REGION Network 12
   // 读重量
   RUNG wire#powerrail
      #Modbus_Master.Modbus_Master(REQ := wire#w1, MB_ADDR := 3, MODE :=, DATA_ADDR := 40104, DATA_LEN := 2, DATA_PTR := #ST6, DONE =>, BUSY =>, ERROR =>, STATUS =>)
      Move(in := #ST6[0], out1 => #B管道内径AT[1])
      Move(in := #ST6[1], out1 => #B管道内径AT[0])
   END_RUNG
   RUNG wire#powerrail
      { S7_Templates := "SrcType := Int" } EQ_Contact(in1 := #CTU.CV, in2 := 8)
      P_Trig( #TP[8] )
   END_RUNG wire#w1
   // the same network as SCL:
   #_w1 := #CTU.CV = 8;
   #_w2 := #_w1 AND NOT #TP[8];   // rising edge
   #TP[8] := #_w1;
   #Modbus_Master(REQ := #_w2, MB_ADDR := 3, DATA_ADDR := 40104, DATA_LEN := 2, DATA_PTR := #ST6, ENO => #_w3);   // Modbus_Master
   IF #_w3 THEN
       #B管道内径AT[1] := #ST6[0];
       #B管道内径AT[0] := #ST6[1];
   END_IF;
END_REGION
END_FUNCTION_BLOCK

FUNCTION_BLOCK "通信心跳"   // FB46, LAD
{ S7_Optimized_Access := 'TRUE' }
VERSION : 0.1
// stored: AutoNumber true, IsIECCheckEnabled false, IsRetainMemResEnabled false, MemoryReserve 100, SetENOAutomatically false, UDAEnableTagReadback false
   VAR_OUTPUT
      通信失联 : Bool;
   END_VAR
   VAR_IN_OUT
      real_SC输出值 : Real;
      real_FK反馈值 : Real;
      超时时间 : Time := T#30S;
      i : Int;
   END_VAR
   VAR
      t1 : TON_TIME;
      t2 { S7_SetPoint := 'True'} : TON_TIME;
      RT1 : R_TRIG;
      间隔时间 : Time := T#5S;
      SC输出值 : Int;
      FK反馈值 : Int;
   END_VAR
   VAR_TEMP
      TM_FZ : Int;
   END_VAR
BEGIN

REGION Network 2 (SCL)
   // 间隔时间，通针开关
   #TM_FZ:=#FK反馈值;

   #SC输出值 := REAL_TO_INT(#real_SC输出值);
   #FK反馈值 := REAL_TO_INT(#real_FK反馈值);

   #t1(IN := (#TM_FZ <> #SC输出值) ,
       PT := #超时时间,
       Q=>#通信失联);


   (* IF #t1.Q THEN
       (* #TM_FZ := 1; *)
       #SC输出值 := #SC输出值 - 1;
   END_IF; *)

   IF #TM_FZ =#SC输出值 THEN

       IF #SC输出值 MOD 2 =0 THEN

           #SC输出值 := #SC输出值 + 1;
       ELSE

           #SC输出值 := #SC输出值 - 1;
       END_IF;

   END_IF;
END_REGION
END_FUNCTION_BLOCK

FUNCTION_BLOCK "52普通脉冲"   // FB23, SCL
{ S7_Optimized_Access := 'TRUE' }
VERSION : 0.1
// stored: AutoNumber true, IsIECCheckEnabled false, IsRetainMemResEnabled false, MemoryReserve 100, SetENOAutomatically false, UDAEnableTagReadback false
   VAR_INPUT
      模式设定 : Real;
      QD : Bool;
      On_Time : Real;
      Stop_Time : Real;
      Num : Int;
   END_VAR
   VAR_OUTPUT
      Output_1 : Bool;
      Output_2 : Bool;
      Output_3 : Bool;
      Output_4 : Bool;
      Output_5 : Bool;
      Output_6 : Bool;
      Output_7 : Bool;
      Output_8 : Bool;
      Num_now : Int;
   END_VAR
   VAR
      Stoptime : Time;
      WorkTime : Time;
      TON_ON : Array[1..10] of TON_TIME;
      TON_OFF : Array[1..10] of TON_TIME;
   END_VAR
BEGIN

   IF #模式设定 = 1.0  OR #模式设定 = 2.0  THEN
       #Stoptime := DINT_TO_TIME(REAL_TO_DINT(#Stop_Time * 1000.0));
       //#WorkTime := DINT_TO_TIME(REAL_TO_DINT(#On_Time * 1000));
        #WorkTime := REAL_TO_DINT(#On_Time);

       IF NOT #QD THEN
           #Num_now := 0;
       ELSE

           IF #Num <= 8 THEN
               #Num_now := #Num;
           ELSE
               #Num_now := 8;
           END_IF;

       END_IF;



       CASE #Num_now OF
           1:
               #TON_ON[1](IN := #QD AND NOT #TON_OFF[1].Q,
                          PT := #WorkTime);
               #TON_OFF[1](IN := #QD AND #TON_ON[1].Q,
                           PT := #Stoptime);


               #Output_1 := #QD AND NOT #TON_ON[1].Q;


           2:  // Statement section case 1
               #TON_ON[1](IN := #QD AND NOT #TON_OFF[2].Q,
                          PT := #WorkTime);
               #TON_OFF[1](IN := #QD AND #TON_ON[1].Q,
                           PT := #Stoptime);
               #TON_ON[2](IN := #QD AND #TON_ON[1].Q AND #TON_OFF[1].Q,
                          PT := #WorkTime);
               #TON_OFF[2](IN := #QD AND #TON_ON[1].Q AND #TON_OFF[1].Q AND #TON_ON[2].Q,
                           PT := #Stoptime);

               #Output_1 := #QD AND NOT #TON_ON[1].Q;
               #Output_2 := #QD AND #TON_ON[1].Q AND #TON_OFF[1].Q AND NOT #TON_ON[2].Q;

           3:  // Statement section case 2 to 4
               #TON_ON[1](IN := #QD AND NOT #TON_OFF[3].Q,
                          PT := #WorkTime);
               #TON_OFF[1](IN := #QD AND #TON_ON[1].Q,
                           PT := #Stoptime);
               #TON_ON[2](IN := #QD AND #TON_ON[1].Q AND #TON_OFF[1].Q,
                          PT := #WorkTime);
               #TON_OFF[2](IN := #QD AND #TON_ON[1].Q AND #TON_OFF[1].Q AND #TON_ON[2].Q,
                           PT := #Stoptime);
               #TON_ON[3](IN := #QD AND #TON_ON[1].Q AND #TON_OFF[1].Q AND #TON_ON[2].Q AND #TON_OFF[2].Q,
                          PT := #WorkTime);
               #TON_OFF[3](IN := #QD AND #TON_ON[1].Q AND #TON_OFF[1].Q AND #TON_ON[2].Q AND #TON_OFF[2].Q AND #TON_ON[3].Q,
                           PT := #Stoptime);
               #Output_1 := #QD AND NOT #TON_ON[1].Q;
               #Output_2 := #QD AND #TON_ON[1].Q AND #TON_OFF[1].Q AND NOT #TON_ON[2].Q;
               #Output_3 := #QD AND #TON_ON[1].Q AND #TON_OFF[1].Q AND #TON_ON[2].Q AND #TON_OFF[2].Q AND NOT #TON_ON[3].Q;
           4:  // Statement section case 2 to 4
               #TON_ON[1](IN := #QD AND NOT #TON_OFF[4].Q,
                          PT := #WorkTime);
               #TON_OFF[1](IN := #QD AND #TON_ON[1].Q,
                           PT := #Stoptime);
               #TON_ON[2](IN := #QD AND #TON_ON[1].Q AND #TON_OFF[1].Q,
                          PT := #WorkTime);
               #TON_OFF[2](IN := #QD AND #TON_ON[1].Q AND #TON_OFF[1].Q AND #TON_ON[2].Q,
                           PT := #Stoptime);
               #TON_ON[3](IN := #QD AND #TON_ON[1].Q AND #TON_OFF[1].Q AND #TON_ON[2].Q AND #TON_OFF[2].Q,
                          PT := #WorkTime);
               #TON_OFF[3](IN := #QD AND #TON_ON[1].Q AND #TON_OFF[1].Q AND #TON_ON[2].Q AND #TON_OFF[2].Q AND #TON_ON[3].Q,
                           PT := #Stoptime);

               #TON_ON[4](IN := #QD AND #TON_ON[1].Q AND #TON_OFF[1].Q AND #TON_ON[2].Q AND #TON_OFF[2].Q AND #TON_ON[3].Q AND #TON_OFF[3].Q,
                          PT := #WorkTime);
               #TON_OFF[4](IN := #QD AND #TON_ON[1].Q AND #TON_OFF[1].Q AND #TON_ON[2].Q AND #TON_OFF[2].Q AND #TON_ON[3].Q AND #TON_OFF[3].Q AND #TON_ON[4].Q,
                           PT := #Stoptime);


               #Output_1 := #QD AND NOT #TON_ON[1].Q;
               #Output_2 := #QD AND #TON_ON[1].Q AND #TON_OFF[1].Q AND NOT #TON_ON[2].Q;
               #Output_3 := #QD AND #TON_ON[1].Q AND #TON_OFF[1].Q AND #TON_ON[2].Q AND #TON_OFF[2].Q AND NOT #TON_ON[3].Q;
               #Output_4 := #QD AND #TON_ON[1].Q AND #TON_OFF[1].Q AND #TON_ON[2].Q AND #TON_OFF[2].Q AND #TON_ON[3].Q AND #TON_OFF[3].Q AND NOT #TON_ON[4].Q;

           5:  // Statement section case 2 to 4
               #TON_ON[1](IN := #QD AND NOT #TON_OFF[5].Q,
                          PT := #WorkTime);
               #TON_OFF[1](IN := #QD AND #TON_ON[1].Q,
                           PT := #Stoptime);
               #TON_ON[2](IN := #QD AND #TON_ON[1].Q AND #TON_OFF[1].Q,
                          PT := #WorkTime);
               #TON_OFF[2](IN := #QD AND #TON_ON[1].Q AND #TON_OFF[1].Q AND #TON_ON[2].Q,
                           PT := #Stoptime);
               #TON_ON[3](IN := #QD AND #TON_ON[1].Q AND #TON_OFF[1].Q AND #TON_ON[2].Q AND #TON_OFF[2].Q,
                          PT := #WorkTime);
               #TON_OFF[3](IN := #QD AND #TON_ON[1].Q AND #TON_OFF[1].Q AND #TON_ON[2].Q AND #TON_OFF[2].Q AND #TON_ON[3].Q,
                           PT := #Stoptime);

               #TON_ON[4](IN := #QD AND #TON_ON[1].Q AND #TON_OFF[1].Q AND #TON_ON[2].Q AND #TON_OFF[2].Q AND #TON_ON[3].Q AND #TON_OFF[3].Q,
                          PT := #WorkTime);
               #TON_OFF[4](IN := #QD AND #TON_ON[1].Q AND #TON_OFF[1].Q AND #TON_ON[2].Q AND #TON_OFF[2].Q AND #TON_ON[3].Q AND #TON_OFF[3].Q AND #TON_ON[4].Q,
                           PT := #Stoptime);

               #TON_ON[5](IN := #QD AND #TON_ON[1].Q AND #TON_OFF[1].Q AND #TON_ON[2].Q AND #TON_OFF[2].Q AND #TON_ON[3].Q AND #TON_OFF[3].Q AND #TON_ON[4].Q AND #TON_OFF[4].Q,
                          PT := #WorkTime);
               #TON_OFF[5](IN := #QD AND #TON_ON[1].Q AND #TON_OFF[1].Q AND #TON_ON[2].Q AND #TON_OFF[2].Q AND #TON_ON[3].Q AND #TON_OFF[3].Q AND #TON_ON[4].Q AND #TON_OFF[4].Q AND #TON_ON[5].Q,
                           PT := #Stoptime);


               #Output_1 := #QD AND NOT #TON_ON[1].Q;
               #Output_2 := #QD AND #TON_ON[1].Q AND #TON_OFF[1].Q AND NOT #TON_ON[2].Q;
               #Output_3 := #QD AND #TON_ON[1].Q AND #TON_OFF[1].Q AND #TON_ON[2].Q AND #TON_OFF[2].Q AND NOT #TON_ON[3].Q;
               #Output_4 := #QD AND #TON_ON[1].Q AND #TON_OFF[1].Q AND #TON_ON[2].Q AND #TON_OFF[2].Q AND #TON_ON[3].Q AND #TON_OFF[3].Q AND NOT #TON_ON[4].Q;
               #Output_5 := #QD AND #TON_ON[1].Q AND #TON_OFF[1].Q AND #TON_ON[2].Q AND #TON_OFF[2].Q AND #TON_ON[3].Q AND #TON_OFF[3].Q AND #TON_ON[4].Q AND #TON_OFF[4].Q AND NOT #TON_ON[5].Q;

           6:  // Statement section case 2 to 4
               #TON_ON[1](IN := #QD AND NOT #TON_OFF[6].Q,
                          PT := #WorkTime);
               #TON_OFF[1](IN := #QD AND #TON_ON[1].Q,
                           PT := #Stoptime);
               #TON_ON[2](IN := #QD AND #TON_ON[1].Q AND #TON_OFF[1].Q,
                          PT := #WorkTime);
               #TON_OFF[2](IN := #QD AND #TON_ON[1].Q AND #TON_OFF[1].Q AND #TON_ON[2].Q,
                           PT := #Stoptime);
               #TON_ON[3](IN := #QD AND #TON_ON[1].Q AND #TON_OFF[1].Q AND #TON_ON[2].Q AND #TON_OFF[2].Q,
                          PT := #WorkTime);
               #TON_OFF[3](IN := #QD AND #TON_ON[1].Q AND #TON_OFF[1].Q AND #TON_ON[2].Q AND #TON_OFF[2].Q AND #TON_ON[3].Q,
                           PT := #Stoptime);

               #TON_ON[4](IN := #QD AND #TON_ON[1].Q AND #TON_OFF[1].Q AND #TON_ON[2].Q AND #TON_OFF[2].Q AND #TON_ON[3].Q AND #TON_OFF[3].Q,
                          PT := #WorkTime);
               #TON_OFF[4](IN := #QD AND #TON_ON[1].Q AND #TON_OFF[1].Q AND #TON_ON[2].Q AND #TON_OFF[2].Q AND #TON_ON[3].Q AND #TON_OFF[3].Q AND #TON_ON[4].Q,
                           PT := #Stoptime);

               #TON_ON[5](IN := #QD AND #TON_ON[1].Q AND #TON_OFF[1].Q AND #TON_ON[2].Q AND #TON_OFF[2].Q AND #TON_ON[3].Q AND #TON_OFF[3].Q AND #TON_ON[4].Q AND #TON_OFF[4].Q,
                          PT := #WorkTime);
               #TON_OFF[5](IN := #QD AND #TON_ON[1].Q AND #TON_OFF[1].Q AND #TON_ON[2].Q AND #TON_OFF[2].Q AND #TON_ON[3].Q AND #TON_OFF[3].Q AND #TON_ON[4].Q AND #TON_OFF[4].Q AND #TON_ON[5].Q,
                           PT := #Stoptime);

               #TON_ON[6](IN := #QD AND #TON_ON[1].Q AND #TON_OFF[1].Q AND #TON_ON[2].Q AND #TON_OFF[2].Q AND #TON_ON[3].Q AND #TON_OFF[3].Q AND #TON_ON[4].Q AND #TON_OFF[4].Q AND #TON_ON[5].Q AND #TON_OFF[5].Q,
                          PT := #WorkTime);
               #TON_OFF[6](IN := #QD AND #TON_ON[1].Q AND #TON_OFF[1].Q AND #TON_ON[2].Q AND #TON_OFF[2].Q AND #TON_ON[3].Q AND #TON_OFF[3].Q AND #TON_ON[4].Q AND #TON_OFF[4].Q AND #TON_ON[5].Q AND #TON_OFF[5].Q AND #TON_ON[6].Q,
                           PT := #Stoptime);


               #Output_1 := #QD AND NOT #TON_ON[1].Q;
               #Output_2 := #QD AND #TON_ON[1].Q AND #TON_OFF[1].Q AND NOT #TON_ON[2].Q;
               #Output_3 := #QD AND #TON_ON[1].Q AND #TON_OFF[1].Q AND #TON_ON[2].Q AND #TON_OFF[2].Q AND NOT #TON_ON[3].Q;
               #Output_4 := #QD AND #TON_ON[1].Q AND #TON_OFF[1].Q AND #TON_ON[2].Q AND #TON_OFF[2].Q AND #TON_ON[3].Q AND #TON_OFF[3].Q AND NOT #TON_ON[4].Q;
               #Output_5 := #QD AND #TON_ON[1].Q AND #TON_OFF[1].Q AND #TON_ON[2].Q AND #TON_OFF[2].Q AND #TON_ON[3].Q AND #TON_OFF[3].Q AND #TON_ON[4].Q AND #TON_OFF[4].Q AND NOT #TON_ON[5].Q;
               #Output_6 := #QD AND #TON_ON[1].Q AND #TON_OFF[1].Q AND #TON_ON[2].Q AND #TON_OFF[2].Q AND #TON_ON[3].Q AND #TON_OFF[3].Q AND #TON_ON[4].Q AND #TON_OFF[4].Q AND #TON_ON[5].Q AND #TON_OFF[5].Q AND NOT #TON_ON[6].Q;

           7:  // Statement section case 2 to 4
               #TON_ON[1](IN := #QD AND NOT #TON_OFF[7].Q,
                          PT := #WorkTime);
               #TON_OFF[1](IN := #QD AND #TON_ON[1].Q,
                           PT := #Stoptime);
               #TON_ON[2](IN := #QD AND #TON_ON[1].Q AND #TON_OFF[1].Q,
                          PT := #WorkTime);
               #TON_OFF[2](IN := #QD AND #TON_ON[1].Q AND #TON_OFF[1].Q AND #TON_ON[2].Q,
                           PT := #Stoptime);
               #TON_ON[3](IN := #QD AND #TON_ON[1].Q AND #TON_OFF[1].Q AND #TON_ON[2].Q AND #TON_OFF[2].Q,
                          PT := #WorkTime);
               #TON_OFF[3](IN := #QD AND #TON_ON[1].Q AND #TON_OFF[1].Q AND #TON_ON[2].Q AND #TON_OFF[2].Q AND #TON_ON[3].Q,
                           PT := #Stoptime);

               #TON_ON[4](IN := #QD AND #TON_ON[1].Q AND #TON_OFF[1].Q AND #TON_ON[2].Q AND #TON_OFF[2].Q AND #TON_ON[3].Q AND #TON_OFF[3].Q,
                          PT := #WorkTime);
               #TON_OFF[4](IN := #QD AND #TON_ON[1].Q AND #TON_OFF[1].Q AND #TON_ON[2].Q AND #TON_OFF[2].Q AND #TON_ON[3].Q AND #TON_OFF[3].Q AND #TON_ON[4].Q,
                           PT := #Stoptime);

               #TON_ON[5](IN := #QD AND #TON_ON[1].Q AND #TON_OFF[1].Q AND #TON_ON[2].Q AND #TON_OFF[2].Q AND #TON_ON[3].Q AND #TON_OFF[3].Q AND #TON_ON[4].Q AND #TON_OFF[4].Q,
                          PT := #WorkTime);
               #TON_OFF[5](IN := #QD AND #TON_ON[1].Q AND #TON_OFF[1].Q AND #TON_ON[2].Q AND #TON_OFF[2].Q AND #TON_ON[3].Q AND #TON_OFF[3].Q AND #TON_ON[4].Q AND #TON_OFF[4].Q AND #TON_ON[5].Q,
                           PT := #Stoptime);

               #TON_ON[6](IN := #QD AND #TON_ON[1].Q AND #TON_OFF[1].Q AND #TON_ON[2].Q AND #TON_OFF[2].Q AND #TON_ON[3].Q AND #TON_OFF[3].Q AND #TON_ON[4].Q AND #TON_OFF[4].Q AND #TON_ON[5].Q AND #TON_OFF[5].Q,
                          PT := #WorkTime);
               #TON_OFF[6](IN := #QD AND #TON_ON[1].Q AND #TON_OFF[1].Q AND #TON_ON[2].Q AND #TON_OFF[2].Q AND #TON_ON[3].Q AND #TON_OFF[3].Q AND #TON_ON[4].Q AND #TON_OFF[4].Q AND #TON_ON[5].Q AND #TON_OFF[5].Q AND #TON_ON[6].Q,
                           PT := #Stoptime);

               #TON_ON[7](IN := #QD AND #TON_ON[1].Q AND #TON_OFF[1].Q AND #TON_ON[2].Q AND #TON_OFF[2].Q AND #TON_ON[3].Q AND #TON_OFF[3].Q AND #TON_ON[4].Q AND #TON_OFF[5].Q AND #TON_ON[5].Q AND #TON_OFF[6].Q AND #TON_ON[6].Q AND #TON_OFF[6].Q,
                          PT := #WorkTime);
               #TON_OFF[7](IN := #QD AND #TON_ON[1].Q AND #TON_OFF[1].Q AND #TON_ON[2].Q AND #TON_OFF[2].Q AND #TON_ON[3].Q AND #TON_OFF[3].Q AND #TON_ON[4].Q AND #TON_OFF[5].Q AND #TON_ON[5].Q AND #TON_OFF[6].Q AND #TON_ON[6].Q AND #TON_OFF[6].Q AND #TON_ON[7].Q,
                           PT := #Stoptime);



               #Output_1 := #QD AND NOT #TON_ON[1].Q;
               #Output_2 := #QD AND #TON_ON[1].Q AND #TON_OFF[1].Q AND NOT #TON_ON[2].Q;
               #Output_3 := #QD AND #TON_ON[1].Q AND #TON_OFF[1].Q AND #TON_ON[2].Q AND #TON_OFF[2].Q AND NOT #TON_ON[3].Q;
               #Output_4 := #QD AND #TON_ON[1].Q AND #TON_OFF[1].Q AND #TON_ON[2].Q AND #TON_OFF[2].Q AND #TON_ON[3].Q AND #TON_OFF[3].Q AND NOT #TON_ON[4].Q;
               #Output_5 := #QD AND #TON_ON[1].Q AND #TON_OFF[1].Q AND #TON_ON[2].Q AND #TON_OFF[2].Q AND #TON_ON[3].Q AND #TON_OFF[3].Q AND #TON_ON[4].Q AND #TON_OFF[4].Q AND NOT #TON_ON[5].Q;
               #Output_6 := #QD AND #TON_ON[1].Q AND #TON_OFF[1].Q AND #TON_ON[2].Q AND #TON_OFF[2].Q AND #TON_ON[3].Q AND #TON_OFF[3].Q AND #TON_ON[4].Q AND #TON_OFF[4].Q AND #TON_ON[5].Q AND #TON_OFF[5].Q AND NOT #TON_ON[6].Q;
               #Output_7 := #QD AND #TON_ON[1].Q AND #TON_OFF[1].Q AND #TON_ON[2].Q AND #TON_OFF[2].Q AND #TON_ON[3].Q AND #TON_OFF[3].Q AND #TON_ON[4].Q AND #TON_OFF[4].Q AND #TON_ON[5].Q AND #TON_OFF[5].Q AND #TON_ON[6].Q AND #TON_OFF[6].Q AND NOT #TON_ON[7].Q;

           8:  // Statement section case 2 to 4
               #TON_ON[1](IN := #QD AND NOT #TON_OFF[8].Q,
                          PT := #WorkTime);
               #TON_OFF[1](IN := #QD AND #TON_ON[1].Q,
                           PT := #Stoptime);
               #TON_ON[2](IN := #QD AND #TON_ON[1].Q AND #TON_OFF[1].Q,
                          PT := #WorkTime);
               #TON_OFF[2](IN := #QD AND #TON_ON[1].Q AND #TON_OFF[1].Q AND #TON_ON[2].Q,
                           PT := #Stoptime);
               #TON_ON[3](IN := #QD AND #TON_ON[1].Q AND #TON_OFF[1].Q AND #TON_ON[2].Q AND #TON_OFF[2].Q,
                          PT := #WorkTime);
               #TON_OFF[3](IN := #QD AND #TON_ON[1].Q AND #TON_OFF[1].Q AND #TON_ON[2].Q AND #TON_OFF[2].Q AND #TON_ON[3].Q,
                           PT := #Stoptime);

               #TON_ON[4](IN := #QD AND #TON_ON[1].Q AND #TON_OFF[1].Q AND #TON_ON[2].Q AND #TON_OFF[2].Q AND #TON_ON[3].Q AND #TON_OFF[3].Q,
                          PT := #WorkTime);
               #TON_OFF[4](IN := #QD AND #TON_ON[1].Q AND #TON_OFF[1].Q AND #TON_ON[2].Q AND #TON_OFF[2].Q AND #TON_ON[3].Q AND #TON_OFF[3].Q AND #TON_ON[4].Q,
                           PT := #Stoptime);

               #TON_ON[5](IN := #QD AND #TON_ON[1].Q AND #TON_OFF[1].Q AND #TON_ON[2].Q AND #TON_OFF[2].Q AND #TON_ON[3].Q AND #TON_OFF[3].Q AND #TON_ON[4].Q AND #TON_OFF[4].Q,
                          PT := #WorkTime);
               #TON_OFF[5](IN := #QD AND #TON_ON[1].Q AND #TON_OFF[1].Q AND #TON_ON[2].Q AND #TON_OFF[2].Q AND #TON_ON[3].Q AND #TON_OFF[3].Q AND #TON_ON[4].Q AND #TON_OFF[4].Q AND #TON_ON[5].Q,
                           PT := #Stoptime);

               #TON_ON[6](IN := #QD AND #TON_ON[1].Q AND #TON_OFF[1].Q AND #TON_ON[2].Q AND #TON_OFF[2].Q AND #TON_ON[3].Q AND #TON_OFF[3].Q AND #TON_ON[4].Q AND #TON_OFF[4].Q AND #TON_ON[5].Q AND #TON_OFF[5].Q,
                          PT := #WorkTime);
               #TON_OFF[6](IN := #QD AND #TON_ON[1].Q AND #TON_OFF[1].Q AND #TON_ON[2].Q AND #TON_OFF[2].Q AND #TON_ON[3].Q AND #TON_OFF[3].Q AND #TON_ON[4].Q AND #TON_OFF[4].Q AND #TON_ON[5].Q AND #TON_OFF[5].Q AND #TON_ON[6].Q,
                           PT := #Stoptime);

               #TON_ON[7](IN := #QD AND #TON_ON[1].Q AND #TON_OFF[1].Q AND #TON_ON[2].Q AND #TON_OFF[2].Q AND #TON_ON[3].Q AND #TON_OFF[3].Q AND #TON_ON[4].Q AND #TON_OFF[4].Q AND #TON_ON[5].Q AND #TON_OFF[5].Q AND #TON_ON[6].Q AND #TON_OFF[6].Q,
                          PT := #WorkTime);
               #TON_OFF[7](IN := #QD AND #TON_ON[1].Q AND #TON_OFF[1].Q AND #TON_ON[2].Q AND #TON_OFF[2].Q AND #TON_ON[3].Q AND #TON_OFF[3].Q AND #TON_ON[4].Q AND #TON_OFF[4].Q AND #TON_ON[5].Q AND #TON_OFF[5].Q AND #TON_ON[6].Q AND #TON_OFF[6].Q AND #TON_ON[7].Q,
                           PT := #Stoptime);
               #TON_ON[8](IN := #QD AND #TON_ON[1].Q AND #TON_OFF[1].Q AND #TON_ON[2].Q AND #TON_OFF[2].Q AND #TON_ON[3].Q AND #TON_OFF[3].Q AND #TON_ON[4].Q AND #TON_OFF[4].Q AND #TON_ON[5].Q AND #TON_OFF[5].Q AND #TON_ON[6].Q AND #TON_OFF[6].Q AND #TON_ON[7].Q AND #TON_OFF[7].Q,
                          PT := #WorkTime);
               #TON_OFF[8](IN := #QD AND #TON_ON[1].Q AND #TON_OFF[1].Q AND #TON_ON[2].Q AND #TON_OFF[2].Q AND #TON_ON[3].Q AND #TON_OFF[3].Q AND #TON_ON[4].Q AND #TON_OFF[4].Q AND #TON_ON[5].Q AND #TON_OFF[5].Q AND #TON_ON[6].Q AND #TON_OFF[6].Q AND #TON_ON[7].Q AND #TON_OFF[7].Q AND #TON_ON[8].Q,
                           PT := #Stoptime);


               #Output_1 := #QD AND NOT #TON_ON[1].Q;
               #Output_2 := #QD AND #TON_ON[1].Q AND #TON_OFF[1].Q AND NOT #TON_ON[2].Q;
               #Output_3 := #QD AND #TON_ON[1].Q AND #TON_OFF[1].Q AND #TON_ON[2].Q AND #TON_OFF[2].Q AND NOT #TON_ON[3].Q;
               #Output_4 := #QD AND #TON_ON[1].Q AND #TON_OFF[1].Q AND #TON_ON[2].Q AND #TON_OFF[2].Q AND #TON_ON[3].Q AND #TON_OFF[3].Q AND NOT #TON_ON[4].Q;
               #Output_5 := #QD AND #TON_ON[1].Q AND #TON_OFF[1].Q AND #TON_ON[2].Q AND #TON_OFF[2].Q AND #TON_ON[3].Q AND #TON_OFF[3].Q AND #TON_ON[4].Q AND #TON_OFF[4].Q AND NOT #TON_ON[5].Q;
               #Output_6 := #QD AND #TON_ON[1].Q AND #TON_OFF[1].Q AND #TON_ON[2].Q AND #TON_OFF[2].Q AND #TON_ON[3].Q AND #TON_OFF[3].Q AND #TON_ON[4].Q AND #TON_OFF[4].Q AND #TON_ON[5].Q AND #TON_OFF[5].Q AND NOT #TON_ON[6].Q;
               #Output_7 := #QD AND #TON_ON[1].Q AND #TON_OFF[1].Q AND #TON_ON[2].Q AND #TON_OFF[2].Q AND #TON_ON[3].Q AND #TON_OFF[3].Q AND #TON_ON[4].Q AND #TON_OFF[4].Q AND #TON_ON[5].Q AND #TON_OFF[5].Q AND #TON_ON[6].Q AND #TON_OFF[6].Q AND NOT #TON_ON[7].Q;
               #Output_8 := #QD AND #TON_ON[1].Q AND #TON_OFF[1].Q AND #TON_ON[2].Q AND #TON_OFF[2].Q AND #TON_ON[3].Q AND #TON_OFF[3].Q AND #TON_ON[4].Q AND #TON_OFF[4].Q AND #TON_ON[5].Q AND #TON_OFF[5].Q AND #TON_ON[6].Q AND #TON_OFF[6].Q AND #TON_ON[7].Q AND #TON_OFF[7].Q AND NOT #TON_ON[8].Q;

           ELSE  // Statement section ELSE
               ;
       END_CASE;
   END_IF;


   IF NOT #QD THEN

       #Output_1 := 0;
       #Output_2 := 0;
       #Output_3 := 0;
       #Output_4 := 0;
       #Output_5 := 0;
       #Output_6 := 0;
       #Output_7 := 0;
       #Output_8 := 0;
   END_IF;
END_FUNCTION_BLOCK

FUNCTION_BLOCK "10-REAL-TIME"   // FB63, LAD
{ S7_Optimized_Access := 'TRUE' }
VERSION : 0.1
// stored: AutoNumber true, IsIECCheckEnabled false, IsRetainMemResEnabled false, MemoryReserve 100, SetENOAutomatically false, UDAEnableTagReadback false
   VAR_INPUT
      时间_Real { ExternalAccessible := 'False'; ExternalVisible := 'False'; ExternalWritable := 'False'} : Real;   // 单位：秒
   END_VAR
   VAR_OUTPUT
      时间_Time { ExternalAccessible := 'False'; ExternalVisible := 'False'; ExternalWritable := 'False'} : Time;
   END_VAR
   VAR_TEMP
      Dint_Temp : DInt;
   END_VAR
BEGIN

REGION Network 1 (SCL)
   #时间_Time := DINT_TO_TIME(REAL_TO_DINT(#时间_Real * 1000.0));
END_REGION
END_FUNCTION_BLOCK

FUNCTION_BLOCK "10-模拟量输入"   // FB40, SCL
{ S7_Optimized_Access := 'TRUE' }
VERSION : 0.1
// stored: AutoNumber true, IsIECCheckEnabled false, IsRetainMemResEnabled false, MemoryReserve 100, SetENOAutomatically false, UDAEnableTagReadback false
   VAR_INPUT
      HMI上限 : Real;
      HMI下限 : Real;
      PLC上限 : Int := 27648;
      PLC下限 : Int;
   END_VAR
   VAR_IN_OUT
      "PLC-仪表" : Int;
      HMI仪表 : Real;
   END_VAR
   VAR
      DBD28 : Real;
   END_VAR
BEGIN
   #DBD28 := NORM_X_REAL(MIN := #PLC下限, VALUE := #"PLC-仪表", MAX := #PLC上限);
   #HMI仪表 := SCALE_X_REAL(MIN := #HMI下限, VALUE := #DBD28, MAX := #HMI上限);
END_FUNCTION_BLOCK

FUNCTION_BLOCK "11-模拟量输出"   // FB55, SCL
{ S7_Optimized_Access := 'TRUE' }
VERSION : 0.1
// stored: AutoNumber true, IsIECCheckEnabled false, IsRetainMemResEnabled false, MemoryReserve 100, SetENOAutomatically false, UDAEnableTagReadback false
   VAR_INPUT
      HMI上限 : Real;
      HMI下限 : Real;
      PLC上限 : Int;
      PLC下限 : Int;
   END_VAR
   VAR_IN_OUT
      PLC调控 : Int;
      HMI设定 : Real;
   END_VAR
   VAR
      DBD1 : Real;
   END_VAR
BEGIN
   #DBD1 := NORM_X_REAL(MIN := #HMI下限, VALUE := #HMI设定, MAX := #HMI上限);
   #PLC调控 := SCALE_X_INT(MIN := #PLC下限, VALUE := #DBD1, MAX := #PLC上限);
END_FUNCTION_BLOCK

FUNCTION_BLOCK "12-2点斜率输入->输出"   // FB41, LAD
{ S7_Optimized_Access := 'TRUE' }
VERSION : 0.1
// stored: AutoNumber true, IsIECCheckEnabled false, IsRetainMemResEnabled false, MemoryReserve 100, SetENOAutomatically false, UDAEnableTagReadback false
   VAR_INPUT
      sr输入ok : Real;
   END_VAR
   VAR_OUTPUT
      sc输出ok : Int;
   END_VAR
   VAR_IN_OUT
      sr输入1 : Real;
      sc输出1 : Real;
      sr输入2 : Real;
      sc输出2 : Real;
   END_VAR
BEGIN

REGION Network 1 (SCL)


   #sc输出ok := REAL_TO_INT(((#sc输出2 - #sc输出1) / (#sr输入2 - #sr输入1)) * #sr输入ok);
END_REGION
END_FUNCTION_BLOCK

FUNCTION_BLOCK "12-2点斜率输出->输入"   // FB54, LAD
{ S7_Optimized_Access := 'TRUE' }
VERSION : 0.1
// stored: AutoNumber true, IsIECCheckEnabled false, IsRetainMemResEnabled false, MemoryReserve 100, SetENOAutomatically false, UDAEnableTagReadback false
   VAR_INPUT
      sc输出ok : Int;
   END_VAR
   VAR_OUTPUT
      sr输入ok : Real;
   END_VAR
   VAR_IN_OUT
      sr输入1 : Real;
      sc输出1 : Real;
      sr输入2 : Real;
      sc输出2 : Real;
   END_VAR
BEGIN

REGION Network 1 (SCL)


   #sr输入ok := REAL_TO_INT(((#sr输入2 - #sr输入1)/(#sc输出2 - #sc输出1) ) * #sc输出ok);
END_REGION
END_FUNCTION_BLOCK

FUNCTION_BLOCK "15-称重系统"   // FB47, LAD
{ S7_Optimized_Access := 'TRUE' }
VERSION : 0.1
// stored: AutoNumber true, IsIECCheckEnabled false, IsRetainMemResEnabled false, MemoryReserve 100, SetENOAutomatically false, UDAEnableTagReadback false
   VAR_OUTPUT
      管道已堵塞 : Bool;
   END_VAR
   VAR_IN_OUT
      PLUS_1S : Bool;
      YX允许值 : Int;
      超时时间 : Time := T#30S;
      FK反馈值 : Int;
      FK初次反馈值 : Int;
      FK二次反馈值 : Int;
      i : UDInt;
      TTIME : Time;
   END_VAR
   VAR
      t1 : TON_TIME;
      RT1 : R_TRIG;
      RT2 : R_TRIG;
      CZ差值 : Int;
      TT : IEC_TIMER;
   END_VAR
   VAR_TEMP
      TM_FZ : Bool;
      j : Int;
   END_VAR
BEGIN

REGION Network 1 (SCL)
   // 间隔时间，通针开关

   #t1(IN := (#CZ差值> #YX允许值) ,
       PT := #超时时间,
       Q=>#管道已堵塞);
   #TTIME := #t1.ET;

   #RT1(CLK := "Clock_1Hz");

   IF  #RT1.Q THEN
       #i += 1;
   END_IF;

   IF #i >= 60 THEN
       #i := 0;
   END_IF;

   IF #i > 0 AND #i < 30 THEN
       #FK初次反馈值 := #FK反馈值;
   END_IF;

   IF #i < 60 AND #i > 30 THEN
       #FK二次反馈值 := #FK反馈值;
   END_IF;

   #CZ差值 := ABS(#FK初次反馈值 - #FK二次反馈值);
END_REGION
END_FUNCTION_BLOCK

FUNCTION_BLOCK "16-普通脉冲"   // FB53, SCL
{ S7_Optimized_Access := 'TRUE' }
VERSION : 0.1
// stored: AutoNumber true, IsIECCheckEnabled false, IsRetainMemResEnabled false, MemoryReserve 100, SetENOAutomatically false, UDAEnableTagReadback false
   VAR_INPUT
      模式设定 : Real;
      QD : Bool;
      On_Time : Real;
      Stop_Time : Real;
      Num : Int;
   END_VAR
   VAR_OUTPUT
      Output_1 : Bool;
      Output_2 : Bool;
      Output_3 : Bool;
      Output_4 : Bool;
      Output_5 : Bool;
      Output_6 : Bool;
      Output_7 : Bool;
      Output_8 : Bool;
      Num_now : Int;
   END_VAR
   VAR
      Stoptime : Time;
      WorkTime : Time;
      TON_ON : Array[1..10] of TON_TIME;
      TON_OFF : Array[1..10] of TON_TIME;
   END_VAR
BEGIN

   IF #模式设定 = 1.0  OR #模式设定 = 2.0  THEN
       #Stoptime := DINT_TO_TIME(REAL_TO_DINT(#Stop_Time * 1000.0));
       //#WorkTime := DINT_TO_TIME(REAL_TO_DINT(#On_Time * 1000));
        #WorkTime := REAL_TO_DINT(#On_Time);

       IF NOT #QD THEN
           #Num_now := 0;
       ELSE

           IF #Num <= 12 THEN
               #Num_now := #Num;
           ELSE
               #Num_now := 12;
           END_IF;

       END_IF;



       CASE #Num_now OF
           1:
               #TON_ON[1](IN := #QD AND NOT #TON_OFF[1].Q,
                          PT := #WorkTime);
               #TON_OFF[1](IN := #QD AND #TON_ON[1].Q,
                           PT := #Stoptime);


               #Output_1 := #QD AND NOT #TON_ON[1].Q;


           2:  // Statement section case 1
               #TON_ON[1](IN := #QD AND NOT #TON_OFF[2].Q,
                          PT := #WorkTime);
               #TON_OFF[1](IN := #QD AND #TON_ON[1].Q,
                           PT := #Stoptime);
               #TON_ON[2](IN := #QD AND #TON_ON[1].Q AND #TON_OFF[1].Q,
                          PT := #WorkTime);
               #TON_OFF[2](IN := #QD AND #TON_ON[1].Q AND #TON_OFF[1].Q AND #TON_ON[2].Q,
                           PT := #Stoptime);

               #Output_1 := #QD AND NOT #TON_ON[1].Q;
               #Output_2 := #QD AND #TON_ON[1].Q AND #TON_OFF[1].Q AND NOT #TON_ON[2].Q;

           3:  // Statement section case 2 to 4
               #TON_ON[1](IN := #QD AND NOT #TON_OFF[3].Q,
                          PT := #WorkTime);
               #TON_OFF[1](IN := #QD AND #TON_ON[1].Q,
                           PT := #Stoptime);
               #TON_ON[2](IN := #QD AND #TON_ON[1].Q AND #TON_OFF[1].Q,
                          PT := #WorkTime);
               #TON_OFF[2](IN := #QD AND #TON_ON[1].Q AND #TON_OFF[1].Q AND #TON_ON[2].Q,
                           PT := #Stoptime);
               #TON_ON[3](IN := #QD AND #TON_ON[1].Q AND #TON_OFF[1].Q AND #TON_ON[2].Q AND #TON_OFF[2].Q,
                          PT := #WorkTime);
               #TON_OFF[3](IN := #QD AND #TON_ON[1].Q AND #TON_OFF[1].Q AND #TON_ON[2].Q AND #TON_OFF[2].Q AND #TON_ON[3].Q,
                           PT := #Stoptime);
               #Output_1 := #QD AND NOT #TON_ON[1].Q;
               #Output_2 := #QD AND #TON_ON[1].Q AND #TON_OFF[1].Q AND NOT #TON_ON[2].Q;
               #Output_3 := #QD AND #TON_ON[1].Q AND #TON_OFF[1].Q AND #TON_ON[2].Q AND #TON_OFF[2].Q AND NOT #TON_ON[3].Q;
           4:  // Statement section case 2 to 4
               #TON_ON[1](IN := #QD AND NOT #TON_OFF[4].Q,
                          PT := #WorkTime);
               #TON_OFF[1](IN := #QD AND #TON_ON[1].Q,
                           PT := #Stoptime);
               #TON_ON[2](IN := #QD AND #TON_ON[1].Q AND #TON_OFF[1].Q,
                          PT := #WorkTime);
               #TON_OFF[2](IN := #QD AND #TON_ON[1].Q AND #TON_OFF[1].Q AND #TON_ON[2].Q,
                           PT := #Stoptime);
               #TON_ON[3](IN := #QD AND #TON_ON[1].Q AND #TON_OFF[1].Q AND #TON_ON[2].Q AND #TON_OFF[2].Q,
                          PT := #WorkTime);
               #TON_OFF[3](IN := #QD AND #TON_ON[1].Q AND #TON_OFF[1].Q AND #TON_ON[2].Q AND #TON_OFF[2].Q AND #TON_ON[3].Q,
                           PT := #Stoptime);

               #TON_ON[4](IN := #QD AND #TON_ON[1].Q AND #TON_OFF[1].Q AND #TON_ON[2].Q AND #TON_OFF[2].Q AND #TON_ON[3].Q AND #TON_OFF[3].Q,
                          PT := #WorkTime);
               #TON_OFF[4](IN := #QD AND #TON_ON[1].Q AND #TON_OFF[1].Q AND #TON_ON[2].Q AND #TON_OFF[2].Q AND #TON_ON[3].Q AND #TON_OFF[3].Q AND #TON_ON[4].Q,
                           PT := #Stoptime);


               #Output_1 := #QD AND NOT #TON_ON[1].Q;
               #Output_2 := #QD AND #TON_ON[1].Q AND #TON_OFF[1].Q AND NOT #TON_ON[2].Q;
               #Output_3 := #QD AND #TON_ON[1].Q AND #TON_OFF[1].Q AND #TON_ON[2].Q AND #TON_OFF[2].Q AND NOT #TON_ON[3].Q;
               #Output_4 := #QD AND #TON_ON[1].Q AND #TON_OFF[1].Q AND #TON_ON[2].Q AND #TON_OFF[2].Q AND #TON_ON[3].Q AND #TON_OFF[3].Q AND NOT #TON_ON[4].Q;

           5:  // Statement section case 2 to 4
               #TON_ON[1](IN := #QD AND NOT #TON_OFF[5].Q,
                          PT := #WorkTime);
               #TON_OFF[1](IN := #QD AND #TON_ON[1].Q,
                           PT := #Stoptime);
               #TON_ON[2](IN := #QD AND #TON_ON[1].Q AND #TON_OFF[1].Q,
                          PT := #WorkTime);
               #TON_OFF[2](IN := #QD AND #TON_ON[1].Q AND #TON_OFF[1].Q AND #TON_ON[2].Q,
                           PT := #Stoptime);
               #TON_ON[3](IN := #QD AND #TON_ON[1].Q AND #TON_OFF[1].Q AND #TON_ON[2].Q AND #TON_OFF[2].Q,
                          PT := #WorkTime);
               #TON_OFF[3](IN := #QD AND #TON_ON[1].Q AND #TON_OFF[1].Q AND #TON_ON[2].Q AND #TON_OFF[2].Q AND #TON_ON[3].Q,
                           PT := #Stoptime);

               #TON_ON[4](IN := #QD AND #TON_ON[1].Q AND #TON_OFF[1].Q AND #TON_ON[2].Q AND #TON_OFF[2].Q AND #TON_ON[3].Q AND #TON_OFF[3].Q,
                          PT := #WorkTime);
               #TON_OFF[4](IN := #QD AND #TON_ON[1].Q AND #TON_OFF[1].Q AND #TON_ON[2].Q AND #TON_OFF[2].Q AND #TON_ON[3].Q AND #TON_OFF[3].Q AND #TON_ON[4].Q,
                           PT := #Stoptime);

               #TON_ON[5](IN := #QD AND #TON_ON[1].Q AND #TON_OFF[1].Q AND #TON_ON[2].Q AND #TON_OFF[2].Q AND #TON_ON[3].Q AND #TON_OFF[3].Q AND #TON_ON[4].Q AND #TON_OFF[4].Q,
                          PT := #WorkTime);
               #TON_OFF[5](IN := #QD AND #TON_ON[1].Q AND #TON_OFF[1].Q AND #TON_ON[2].Q AND #TON_OFF[2].Q AND #TON_ON[3].Q AND #TON_OFF[3].Q AND #TON_ON[4].Q AND #TON_OFF[4].Q AND #TON_ON[5].Q,
                           PT := #Stoptime);


               #Output_1 := #QD AND NOT #TON_ON[1].Q;
               #Output_2 := #QD AND #TON_ON[1].Q AND #TON_OFF[1].Q AND NOT #TON_ON[2].Q;
               #Output_3 := #QD AND #TON_ON[1].Q AND #TON_OFF[1].Q AND #TON_ON[2].Q AND #TON_OFF[2].Q AND NOT #TON_ON[3].Q;
               #Output_4 := #QD AND #TON_ON[1].Q AND #TON_OFF[1].Q AND #TON_ON[2].Q AND #TON_OFF[2].Q AND #TON_ON[3].Q AND #TON_OFF[3].Q AND NOT #TON_ON[4].Q;
               #Output_5 := #QD AND #TON_ON[1].Q AND #TON_OFF[1].Q AND #TON_ON[2].Q AND #TON_OFF[2].Q AND #TON_ON[3].Q AND #TON_OFF[3].Q AND #TON_ON[4].Q AND #TON_OFF[4].Q AND NOT #TON_ON[5].Q;

           6:  // Statement section case 2 to 4
               #TON_ON[1](IN := #QD AND NOT #TON_OFF[6].Q,
                          PT := #WorkTime);
               #TON_OFF[1](IN := #QD AND #TON_ON[1].Q,
                           PT := #Stoptime);
               #TON_ON[2](IN := #QD AND #TON_ON[1].Q AND #TON_OFF[1].Q,
                          PT := #WorkTime);
               #TON_OFF[2](IN := #QD AND #TON_ON[1].Q AND #TON_OFF[1].Q AND #TON_ON[2].Q,
                           PT := #Stoptime);
               #TON_ON[3](IN := #QD AND #TON_ON[1].Q AND #TON_OFF[1].Q AND #TON_ON[2].Q AND #TON_OFF[2].Q,
                          PT := #WorkTime);
               #TON_OFF[3](IN := #QD AND #TON_ON[1].Q AND #TON_OFF[1].Q AND #TON_ON[2].Q AND #TON_OFF[2].Q AND #TON_ON[3].Q,
                           PT := #Stoptime);

               #TON_ON[4](IN := #QD AND #TON_ON[1].Q AND #TON_OFF[1].Q AND #TON_ON[2].Q AND #TON_OFF[2].Q AND #TON_ON[3].Q AND #TON_OFF[3].Q,
                          PT := #WorkTime);
               #TON_OFF[4](IN := #QD AND #TON_ON[1].Q AND #TON_OFF[1].Q AND #TON_ON[2].Q AND #TON_OFF[2].Q AND #TON_ON[3].Q AND #TON_OFF[3].Q AND #TON_ON[4].Q,
                           PT := #Stoptime);

               #TON_ON[5](IN := #QD AND #TON_ON[1].Q AND #TON_OFF[1].Q AND #TON_ON[2].Q AND #TON_OFF[2].Q AND #TON_ON[3].Q AND #TON_OFF[3].Q AND #TON_ON[4].Q AND #TON_OFF[4].Q,
                          PT := #WorkTime);
               #TON_OFF[5](IN := #QD AND #TON_ON[1].Q AND #TON_OFF[1].Q AND #TON_ON[2].Q AND #TON_OFF[2].Q AND #TON_ON[3].Q AND #TON_OFF[3].Q AND #TON_ON[4].Q AND #TON_OFF[4].Q AND #TON_ON[5].Q,
                           PT := #Stoptime);

               #TON_ON[6](IN := #QD AND #TON_ON[1].Q AND #TON_OFF[1].Q AND #TON_ON[2].Q AND #TON_OFF[2].Q AND #TON_ON[3].Q AND #TON_OFF[3].Q AND #TON_ON[4].Q AND #TON_OFF[4].Q AND #TON_ON[5].Q AND #TON_OFF[5].Q,
                          PT := #WorkTime);
               #TON_OFF[6](IN := #QD AND #TON_ON[1].Q AND #TON_OFF[1].Q AND #TON_ON[2].Q AND #TON_OFF[2].Q AND #TON_ON[3].Q AND #TON_OFF[3].Q AND #TON_ON[4].Q AND #TON_OFF[4].Q AND #TON_ON[5].Q AND #TON_OFF[5].Q AND #TON_ON[6].Q,
                           PT := #Stoptime);


               #Output_1 := #QD AND NOT #TON_ON[1].Q;
               #Output_2 := #QD AND #TON_ON[1].Q AND #TON_OFF[1].Q AND NOT #TON_ON[2].Q;
               #Output_3 := #QD AND #TON_ON[1].Q AND #TON_OFF[1].Q AND #TON_ON[2].Q AND #TON_OFF[2].Q AND NOT #TON_ON[3].Q;
               #Output_4 := #QD AND #TON_ON[1].Q AND #TON_OFF[1].Q AND #TON_ON[2].Q AND #TON_OFF[2].Q AND #TON_ON[3].Q AND #TON_OFF[3].Q AND NOT #TON_ON[4].Q;
               #Output_5 := #QD AND #TON_ON[1].Q AND #TON_OFF[1].Q AND #TON_ON[2].Q AND #TON_OFF[2].Q AND #TON_ON[3].Q AND #TON_OFF[3].Q AND #TON_ON[4].Q AND #TON_OFF[4].Q AND NOT #TON_ON[5].Q;
               #Output_6 := #QD AND #TON_ON[1].Q AND #TON_OFF[1].Q AND #TON_ON[2].Q AND #TON_OFF[2].Q AND #TON_ON[3].Q AND #TON_OFF[3].Q AND #TON_ON[4].Q AND #TON_OFF[4].Q AND #TON_ON[5].Q AND #TON_OFF[5].Q AND NOT #TON_ON[6].Q;

           7:  // Statement section case 2 to 4
               #TON_ON[1](IN := #QD AND NOT #TON_OFF[7].Q,
                          PT := #WorkTime);
               #TON_OFF[1](IN := #QD AND #TON_ON[1].Q,
                           PT := #Stoptime);
               #TON_ON[2](IN := #QD AND #TON_ON[1].Q AND #TON_OFF[1].Q,
                          PT := #WorkTime);
               #TON_OFF[2](IN := #QD AND #TON_ON[1].Q AND #TON_OFF[1].Q AND #TON_ON[2].Q,
                           PT := #Stoptime);
               #TON_ON[3](IN := #QD AND #TON_ON[1].Q AND #TON_OFF[1].Q AND #TON_ON[2].Q AND #TON_OFF[2].Q,
                          PT := #WorkTime);
               #TON_OFF[3](IN := #QD AND #TON_ON[1].Q AND #TON_OFF[1].Q AND #TON_ON[2].Q AND #TON_OFF[2].Q AND #TON_ON[3].Q,
                           PT := #Stoptime);

               #TON_ON[4](IN := #QD AND #TON_ON[1].Q AND #TON_OFF[1].Q AND #TON_ON[2].Q AND #TON_OFF[2].Q AND #TON_ON[3].Q AND #TON_OFF[3].Q,
                          PT := #WorkTime);
               #TON_OFF[4](IN := #QD AND #TON_ON[1].Q AND #TON_OFF[1].Q AND #TON_ON[2].Q AND #TON_OFF[2].Q AND #TON_ON[3].Q AND #TON_OFF[3].Q AND #TON_ON[4].Q,
                           PT := #Stoptime);

               #TON_ON[5](IN := #QD AND #TON_ON[1].Q AND #TON_OFF[1].Q AND #TON_ON[2].Q AND #TON_OFF[2].Q AND #TON_ON[3].Q AND #TON_OFF[3].Q AND #TON_ON[4].Q AND #TON_OFF[4].Q,
                          PT := #WorkTime);
               #TON_OFF[5](IN := #QD AND #TON_ON[1].Q AND #TON_OFF[1].Q AND #TON_ON[2].Q AND #TON_OFF[2].Q AND #TON_ON[3].Q AND #TON_OFF[3].Q AND #TON_ON[4].Q AND #TON_OFF[4].Q AND #TON_ON[5].Q,
                           PT := #Stoptime);

               #TON_ON[6](IN := #QD AND #TON_ON[1].Q AND #TON_OFF[1].Q AND #TON_ON[2].Q AND #TON_OFF[2].Q AND #TON_ON[3].Q AND #TON_OFF[3].Q AND #TON_ON[4].Q AND #TON_OFF[4].Q AND #TON_ON[5].Q AND #TON_OFF[5].Q,
                          PT := #WorkTime);
               #TON_OFF[6](IN := #QD AND #TON_ON[1].Q AND #TON_OFF[1].Q AND #TON_ON[2].Q AND #TON_OFF[2].Q AND #TON_ON[3].Q AND #TON_OFF[3].Q AND #TON_ON[4].Q AND #TON_OFF[4].Q AND #TON_ON[5].Q AND #TON_OFF[5].Q AND #TON_ON[6].Q,
                           PT := #Stoptime);

               #TON_ON[7](IN := #QD AND #TON_ON[1].Q AND #TON_OFF[1].Q AND #TON_ON[2].Q AND #TON_OFF[2].Q AND #TON_ON[3].Q AND #TON_OFF[3].Q AND #TON_ON[4].Q AND #TON_OFF[5].Q AND #TON_ON[5].Q AND #TON_OFF[6].Q AND #TON_ON[6].Q AND #TON_OFF[6].Q,
                          PT := #WorkTime);
               #TON_OFF[7](IN := #QD AND #TON_ON[1].Q AND #TON_OFF[1].Q AND #TON_ON[2].Q AND #TON_OFF[2].Q AND #TON_ON[3].Q AND #TON_OFF[3].Q AND #TON_ON[4].Q AND #TON_OFF[5].Q AND #TON_ON[5].Q AND #TON_OFF[6].Q AND #TON_ON[6].Q AND #TON_OFF[6].Q AND #TON_ON[7].Q,
                           PT := #Stoptime);



               #Output_1 := #QD AND NOT #TON_ON[1].Q;
               #Output_2 := #QD AND #TON_ON[1].Q AND #TON_OFF[1].Q AND NOT #TON_ON[2].Q;
               #Output_3 := #QD AND #TON_ON[1].Q AND #TON_OFF[1].Q AND #TON_ON[2].Q AND #TON_OFF[2].Q AND NOT #TON_ON[3].Q;
               #Output_4 := #QD AND #TON_ON[1].Q AND #TON_OFF[1].Q AND #TON_ON[2].Q AND #TON_OFF[2].Q AND #TON_ON[3].Q AND #TON_OFF[3].Q AND NOT #TON_ON[4].Q;
               #Output_5 := #QD AND #TON_ON[1].Q AND #TON_OFF[1].Q AND #TON_ON[2].Q AND #TON_OFF[2].Q AND #TON_ON[3].Q AND #TON_OFF[3].Q AND #TON_ON[4].Q AND #TON_OFF[4].Q AND NOT #TON_ON[5].Q;
               #Output_6 := #QD AND #TON_ON[1].Q AND #TON_OFF[1].Q AND #TON_ON[2].Q AND #TON_OFF[2].Q AND #TON_ON[3].Q AND #TON_OFF[3].Q AND #TON_ON[4].Q AND #TON_OFF[4].Q AND #TON_ON[5].Q AND #TON_OFF[5].Q AND NOT #TON_ON[6].Q;
               #Output_7 := #QD AND #TON_ON[1].Q AND #TON_OFF[1].Q AND #TON_ON[2].Q AND #TON_OFF[2].Q AND #TON_ON[3].Q AND #TON_OFF[3].Q AND #TON_ON[4].Q AND #TON_OFF[4].Q AND #TON_ON[5].Q AND #TON_OFF[5].Q AND #TON_ON[6].Q AND #TON_OFF[6].Q AND NOT #TON_ON[7].Q;

           8:  // Statement section case 2 to 4
               #TON_ON[1](IN := #QD AND NOT #TON_OFF[8].Q,
                          PT := #WorkTime);
               #TON_OFF[1](IN := #QD AND #TON_ON[1].Q,
                           PT := #Stoptime);
               #TON_ON[2](IN := #QD AND #TON_ON[1].Q AND #TON_OFF[1].Q,
                          PT := #WorkTime);
               #TON_OFF[2](IN := #QD AND #TON_ON[1].Q AND #TON_OFF[1].Q AND #TON_ON[2].Q,
                           PT := #Stoptime);
               #TON_ON[3](IN := #QD AND #TON_ON[1].Q AND #TON_OFF[1].Q AND #TON_ON[2].Q AND #TON_OFF[2].Q,
                          PT := #WorkTime);
               #TON_OFF[3](IN := #QD AND #TON_ON[1].Q AND #TON_OFF[1].Q AND #TON_ON[2].Q AND #TON_OFF[2].Q AND #TON_ON[3].Q,
                           PT := #Stoptime);

               #TON_ON[4](IN := #QD AND #TON_ON[1].Q AND #TON_OFF[1].Q AND #TON_ON[2].Q AND #TON_OFF[2].Q AND #TON_ON[3].Q AND #TON_OFF[3].Q,
                          PT := #WorkTime);
               #TON_OFF[4](IN := #QD AND #TON_ON[1].Q AND #TON_OFF[1].Q AND #TON_ON[2].Q AND #TON_OFF[2].Q AND #TON_ON[3].Q AND #TON_OFF[3].Q AND #TON_ON[4].Q,
                           PT := #Stoptime);

               #TON_ON[5](IN := #QD AND #TON_ON[1].Q AND #TON_OFF[1].Q AND #TON_ON[2].Q AND #TON_OFF[2].Q AND #TON_ON[3].Q AND #TON_OFF[3].Q AND #TON_ON[4].Q AND #TON_OFF[4].Q,
                          PT := #WorkTime);
               #TON_OFF[5](IN := #QD AND #TON_ON[1].Q AND #TON_OFF[1].Q AND #TON_ON[2].Q AND #TON_OFF[2].Q AND #TON_ON[3].Q AND #TON_OFF[3].Q AND #TON_ON[4].Q AND #TON_OFF[4].Q AND #TON_ON[5].Q,
                           PT := #Stoptime);

               #TON_ON[6](IN := #QD AND #TON_ON[1].Q AND #TON_OFF[1].Q AND #TON_ON[2].Q AND #TON_OFF[2].Q AND #TON_ON[3].Q AND #TON_OFF[3].Q AND #TON_ON[4].Q AND #TON_OFF[4].Q AND #TON_ON[5].Q AND #TON_OFF[5].Q,
                          PT := #WorkTime);
               #TON_OFF[6](IN := #QD AND #TON_ON[1].Q AND #TON_OFF[1].Q AND #TON_ON[2].Q AND #TON_OFF[2].Q AND #TON_ON[3].Q AND #TON_OFF[3].Q AND #TON_ON[4].Q AND #TON_OFF[4].Q AND #TON_ON[5].Q AND #TON_OFF[5].Q AND #TON_ON[6].Q,
                           PT := #Stoptime);

               #TON_ON[7](IN := #QD AND #TON_ON[1].Q AND #TON_OFF[1].Q AND #TON_ON[2].Q AND #TON_OFF[2].Q AND #TON_ON[3].Q AND #TON_OFF[3].Q AND #TON_ON[4].Q AND #TON_OFF[4].Q AND #TON_ON[5].Q AND #TON_OFF[5].Q AND #TON_ON[6].Q AND #TON_OFF[6].Q,
                          PT := #WorkTime);
               #TON_OFF[7](IN := #QD AND #TON_ON[1].Q AND #TON_OFF[1].Q AND #TON_ON[2].Q AND #TON_OFF[2].Q AND #TON_ON[3].Q AND #TON_OFF[3].Q AND #TON_ON[4].Q AND #TON_OFF[4].Q AND #TON_ON[5].Q AND #TON_OFF[5].Q AND #TON_ON[6].Q AND #TON_OFF[6].Q AND #TON_ON[7].Q,
                           PT := #Stoptime);
               #TON_ON[8](IN := #QD AND #TON_ON[1].Q AND #TON_OFF[1].Q AND #TON_ON[2].Q AND #TON_OFF[2].Q AND #TON_ON[3].Q AND #TON_OFF[3].Q AND #TON_ON[4].Q AND #TON_OFF[4].Q AND #TON_ON[5].Q AND #TON_OFF[5].Q AND #TON_ON[6].Q AND #TON_OFF[6].Q AND #TON_ON[7].Q AND #TON_OFF[7].Q,
                          PT := #WorkTime);
               #TON_OFF[8](IN := #QD AND #TON_ON[1].Q AND #TON_OFF[1].Q AND #TON_ON[2].Q AND #TON_OFF[2].Q AND #TON_ON[3].Q AND #TON_OFF[3].Q AND #TON_ON[4].Q AND #TON_OFF[4].Q AND #TON_ON[5].Q AND #TON_OFF[5].Q AND #TON_ON[6].Q AND #TON_OFF[6].Q AND #TON_ON[7].Q AND #TON_OFF[7].Q AND #TON_ON[8].Q,
                           PT := #Stoptime);


               #Output_1 := #QD AND NOT #TON_ON[1].Q;
               #Output_2 := #QD AND #TON_ON[1].Q AND #TON_OFF[1].Q AND NOT #TON_ON[2].Q;
               #Output_3 := #QD AND #TON_ON[1].Q AND #TON_OFF[1].Q AND #TON_ON[2].Q AND #TON_OFF[2].Q AND NOT #TON_ON[3].Q;
               #Output_4 := #QD AND #TON_ON[1].Q AND #TON_OFF[1].Q AND #TON_ON[2].Q AND #TON_OFF[2].Q AND #TON_ON[3].Q AND #TON_OFF[3].Q AND NOT #TON_ON[4].Q;
               #Output_5 := #QD AND #TON_ON[1].Q AND #TON_OFF[1].Q AND #TON_ON[2].Q AND #TON_OFF[2].Q AND #TON_ON[3].Q AND #TON_OFF[3].Q AND #TON_ON[4].Q AND #TON_OFF[4].Q AND NOT #TON_ON[5].Q;
               #Output_6 := #QD AND #TON_ON[1].Q AND #TON_OFF[1].Q AND #TON_ON[2].Q AND #TON_OFF[2].Q AND #TON_ON[3].Q AND #TON_OFF[3].Q AND #TON_ON[4].Q AND #TON_OFF[4].Q AND #TON_ON[5].Q AND #TON_OFF[5].Q AND NOT #TON_ON[6].Q;
               #Output_7 := #QD AND #TON_ON[1].Q AND #TON_OFF[1].Q AND #TON_ON[2].Q AND #TON_OFF[2].Q AND #TON_ON[3].Q AND #TON_OFF[3].Q AND #TON_ON[4].Q AND #TON_OFF[4].Q AND #TON_ON[5].Q AND #TON_OFF[5].Q AND #TON_ON[6].Q AND #TON_OFF[6].Q AND NOT #TON_ON[7].Q;
               #Output_8 := #QD AND #TON_ON[1].Q AND #TON_OFF[1].Q AND #TON_ON[2].Q AND #TON_OFF[2].Q AND #TON_ON[3].Q AND #TON_OFF[3].Q AND #TON_ON[4].Q AND #TON_OFF[4].Q AND #TON_ON[5].Q AND #TON_OFF[5].Q AND #TON_ON[6].Q AND #TON_OFF[6].Q AND #TON_ON[7].Q AND #TON_OFF[7].Q AND NOT #TON_ON[8].Q;

           ELSE  // Statement section ELSE
               ;
       END_CASE;
   END_IF;


   IF NOT #QD THEN

       #Output_1 := 0;
       #Output_2 := 0;
       #Output_3 := 0;
       #Output_4 := 0;
       #Output_5 := 0;
       #Output_6 := 0;
       #Output_7 := 0;
       #Output_8 := 0;
   END_IF;
END_FUNCTION_BLOCK

FUNCTION "GetSymbolName" : WString   // FC910, SCL
TITLE = GetSymbolName
AUTHOR : Siemens
FAMILY : SymInfo
NAME : GetSymNa
VERSION : 1.2
// stored: IsIECCheckEnabled false, SetENOAutomatically false, UDAEnableTagReadback false
   VAR_INPUT
      SymInfo : Variant;
      ParaNr : UInt;
      Size : DInt;
   END_VAR
BEGIN
END_FUNCTION

FUNCTION_BLOCK "MB_CLIENT"   // FB1084, SCL
TITLE = Modbus client communication
AUTHOR : SIMATIC
FAMILY : MBUS_TCP
NAME : MB_CLI
VERSION : 6.0
// stored: IsIECCheckEnabled false, SetENOAutomatically false, UDAEnableTagReadback false
   VAR_INPUT
      REQ : Bool;   // Activates the requested transmission if TRUE
      DISCONNECT : Bool;   // Initiates a disconnect operation
      MB_MODE : USInt;   // Specifies the type of request: read, write or diagnostic
      MB_DATA_ADDR : UDInt;   // Specifies the starting address of the data to be accessed in the Modbus client
      MB_DATA_LEN : UInt;   // Specifies the number of bits or words to be accessed
      RD_MB_DATA_ADDR : UInt;   // Specifies the starting address of the data to be accessed in the Modbus client / Specifies the starting address of the data to be read from the Modbus server
      RD_MB_DATA_LEN : UInt;   // Specifies the number of bits or words to be accessed / Specifies the number of bits or words to be read from the Modbus server
      WR_MB_DATA_ADDR : UInt;   // Specifies the starting address of the data to be accessed in the Modbus client / Specifies the starting address of the data to be written the Modbus server
      WR_MB_DATA_LEN : UInt;   // Specifies the number of bits or words to be accessed / Specifies the number of bits or words to be written to the Modbus server
   END_VAR
   VAR_OUTPUT
      DONE : Bool;   // Instruction finished without error
      BUSY : Bool;   // Modbus transaction in progress
      ERROR : Bool;   // Instruction finished with error
      STATUS { ExternalVisible := 'False'} : Word := 16#0000;   // Detailed error information
   END_VAR
   VAR_IN_OUT
      MB_DATA_PTR : Variant;   // Reference to the local source or destination address
      CONNECT : Variant;   // Reference to the connection parameters
      RD_MB_DATA_PTR : Variant;   // Reference to the memory area to store the data that is to be read from the Modbus server
      WR_MB_DATA_PTR : Variant;   // Reference to the memory area to retrieve the data that is to be written to the Modbus server
   END_VAR
   VAR
      TCON { S7_SetPoint := 'True'} : TCON;   // Local instance of the instruction TCON
      TDISCON { S7_SetPoint := 'True'} : TDISCON;   // Local instance of the instruction TDISCON
      TSEND { S7_SetPoint := 'True'} : TSEND;   // Local instance of the instruction TSEND
      TRECEIVE { S7_SetPoint := 'True'} : TRCV;   // Local instance of the instruction TRCV
      TRESET { S7_SetPoint := 'True'} : T_RESET;   // Local instance of the instruction T_RESET
      TDIAG { S7_SetPoint := 'True'} : T_DIAG;   // Local instance of the instruction T_DIAG
      TDIAG_Status { S7_SetPoint := 'True'} : TDiag_Status;   // TDiag_Status structure
      Blocked_Proc_Timeout : Real := 3.0;   // Time to wait upon a blocked Modbus Client instance before setting inactive
      Rcv_Timeout : Real := 2.0;   // Amount of time that the client waits for the server to respond to a request
      MB_Unit_ID : Byte := 16#FF;   // The MODBUS slave address / The Modbus slave address
      MB_Transaction_ID : Word := 1;   // Number of the current transaction
      RD_MB_DATA_PTR_Length : UDInt;
      WR_MB_DATA_PTR_Length : UDInt;
      MB_State { ExternalWritable := 'False'} : Word;   // Internal state of the Modbus client operation
      SAVED_MB_DATA_ADDR : UDInt;   // For internal use only
      SAVED_DATA_LEN : UInt;   // For internal use only
      SAVED_MB_MODE : USInt;   // For internal use only
      Connection_ID : Word;   // For internal use only
      Retries : Word := 3;   // Number of retries that the client will attempt before returning a no response error
   END_VAR
   VAR DB_SPECIFIC
      TEMP_DATA { ExternalWritable := 'False'} : Array[1..263] of Byte;   // For internal use only
   END_VAR
   VAR
      FC1_4_Req AT TEMP_DATA : TCP_MB_FC1_4_Req;   // For internal use only
      FC1_4_ValResp AT TEMP_DATA : TCP_MB_FC1_4_ValResp;   // For internal use only
      FC5_6_Req AT TEMP_DATA : TCP_MB_FC5_6_Req;   // For internal use only
      FC5_6_ValResp AT TEMP_DATA : TCP_MB_FC5_6_ValResp;   // For internal use only
      FC15_16_Req AT TEMP_DATA : TCP_MB_FC15_16_Req;   // For internal use only
      FC11_Req AT TEMP_DATA : TCP_MB_FC11_Req;   // For internal use only
      FC8_Req AT TEMP_DATA : TCP_MB_FC8_Req;   // For internal use only
      FCx_ErrResp AT TEMP_DATA : TCP_MB_FCx_ErrResp;   // For internal use only
      FC11_ValResp AT TEMP_DATA : Struct
         Transaction_ID : Word;
         Protocol_ID : Word;
         Length : Word;
         Unit_ID : Byte;
         FCode : Byte;
         Data : Array[1..4] of Byte;
      END_STRUCT;
      MB_Buffer_Req AT TEMP_DATA : Struct
         TransactionId : UInt;
         ProtocolId : UInt;
         Length : UInt;
         UID : USInt;
         FCode : USInt;
         Address : UInt;
         Quanity_Value : UInt;
      END_STRUCT;
      MB_Buffer_Resp AT TEMP_DATA : Struct
         TransactionId : UInt;
         ProtocolId : UInt;
         Length : UInt;
         UID : USInt;
         FCode : USInt;
         ByteCount : USInt;
         Data1 : USInt;
         Data : Array[1..252] of Byte;
      END_STRUCT;
      FC23_Req AT TEMP_DATA : Struct
         Transaction_ID : Word;
         Protocol_ID : Word;
         Length : Word;
         Unit_ID : Byte;
         FCode : Byte;
         read_addr : Word;
         read_len : Word;
         write_addr : Word;
         write_len : Word;
         byte_count : Byte;
         Value1 : Byte;
         Values : Array[0..240] of Byte;
      END_STRUCT;
      rcv_timer { ExternalAccessible := 'False'; ExternalVisible := 'False'; ExternalWritable := 'False'; S7_SetPoint := 'True'} : TON_TIME;   // For internal use only
      wd_timer { ExternalAccessible := 'False'; ExternalVisible := 'False'; ExternalWritable := 'False'; S7_SetPoint := 'True'} : TON_TIME;   // For internal use only
      Connected : Bool;   // Connection state
      Active { ExternalWritable := 'False'} : Bool;   // This call is the active instance
      BytesReceived : UDInt;
      Func_Code_23_saved { ExternalAccessible := 'False'; ExternalVisible := 'False'; ExternalWritable := 'False'} : Struct
         mb_data_addr_read { ExternalAccessible := 'False'; ExternalVisible := 'False'; ExternalWritable := 'False'} : Word;
         mb_data_len_read { ExternalAccessible := 'False'; ExternalVisible := 'False'; ExternalWritable := 'False'} : Word;
         mb_data_addr_write { ExternalAccessible := 'False'; ExternalVisible := 'False'; ExternalWritable := 'False'} : Word;
         mb_data_len_write { ExternalAccessible := 'False'; ExternalVisible := 'False'; ExternalWritable := 'False'} : Word;
      END_STRUCT;
   END_VAR
BEGIN
END_FUNCTION_BLOCK

FUNCTION_BLOCK "PID_Compact"   // FB1130, SCL
TITLE = Compact PID_Controller with self-tuning
AUTHOR : SIMATIC
FAMILY : COMPPID
NAME : PID_Cmpt
VERSION : 2.4
// stored: IsIECCheckEnabled false, SetENOAutomatically false, UDAEnableTagReadback false
   VAR_INPUT
      Setpoint : Real;   // controller setpoint input / Sollwerteingang
      Input : Real;   // current value from process in REAL format / Istwert im REAL-Format
      Input_PER : Int;   // current value from peripheral input / Istwert im Peripherieformat
      Disturbance : Real;   // disturbance intrusion / Störaufschaltung
      ManualEnable : Bool;   // activate manual value to overwrite output value / Handwert wird zum Überschreiben des Ausgangswerts aktiviert
      ManualValue : Real;   // manual value / Handwert
      ErrorAck : Bool;   // reset error message / Löschen der Fehlermeldung
      Reset : Bool;   // reset the controller / Rücksetzen, Neustart des Reglers
      ModeActivate : Bool;   // enable mode / Modus freigeben
   END_VAR
   VAR_OUTPUT
      ScaledInput { ExternalWritable := 'False'} : Real;   // current value after scaling / Normierter Istwert
      Output { ExternalWritable := 'False'} : Real;   // output value in REAL format / Ausgangswert im REAL-Format
      Output_PER { ExternalWritable := 'False'} : Int;   // analog output value / Ausgangswert im Peripherieformat
      Output_PWM { ExternalWritable := 'False'} : Bool;   // pulse width modulated output value / Pulsweitenmodulierter Ausgangswert
      SetpointLimit_H { ExternalWritable := 'False'} : Bool;   // setpoint reached upper limit / Oberer Grenzwertmelder Sollwert
      SetpointLimit_L { ExternalWritable := 'False'} : Bool;   // setpoint reached lower limit / Unterer Grenzwertmelder Sollwert
      InputWarning_H { ExternalWritable := 'False'} : Bool;   // current value reached upper warning level / Warnung für Überschreitung der oberen Istwertwarngrenze
      InputWarning_L { ExternalWritable := 'False'} : Bool;   // current value reached lower warning level / Warnung für Unterschreitung der unteren Iswertwarngrenze
      State { ExternalWritable := 'False'} : Int;   // current mode of operation (0-Inactive, 1-SUT, 2-TIR, 3-Automatic, 4-Manual, 5-Substitute output) / Aktuelle Betriebsart (0-Inaktiv, 1-SUT, 2-TIR, 3-Automatik, 4-Hand, 5-Ersatzausgangswert)
      Error { ExternalWritable := 'False'} : Bool;   // error flag / Errorflag
      ErrorBits { ExternalWritable := 'False'} : DWord;   // error message / Fehlermeldung
   END_VAR
   VAR_IN_OUT
      Mode : Int := 4;   // mode selection / Modusanwahl
   END_VAR
   VAR
      InternalDiagnostic : DWord := 0;   // internal diagnostic and version handling / Interne Diagnose und Versionshandling
      InternalVersion { ExternalWritable := 'False'} : DWord := DW#16#02040001;   // version of controller / Version des Reglers
      InternalRTVersion : DWord := 0;   // version of runtime / Version des RunTime
      IntegralResetMode { S7_SetPoint := 'True'} : Int := 4;   // 0 smooth, 1 clear, 2 keep, 3 overwrite initial output, 4 like setpoint change / 0 glätten, 1 löschen, 2 halten, 3 Initialoutput Ablöseregelung, 4 wie Sollwertänderung
      OverwriteInitialOutputValue : Real;   // initialisation of output value for override control / Initialisierungswert des Ausgangswerts für Ablöseregelung
      RunModeByStartup { S7_SetPoint := 'True'} : Bool := true;   // activate Mode after CPU restart / Nach CPU Neustart Mode aktivieren
      LoadBackUp : Bool;   // restore last parameter set / Hochladen des Backupdatensatzes
      SetSubstituteOutput { S7_SetPoint := 'True'} : Bool := true;   // assignment of output value in State = 5 (FALSE - last valid value, TRUE - SubstituteOutput) / Belegung des Ausgangswerts bei State = 5 (FALSE - letzter gültiger Wert, TRUE - Ersatzwert SubstituteOutput)
      PhysicalUnit { ExternalWritable := 'False'; S7_SetPoint := 'True'} : Int;   // unit of measurement of the process value and setpoint / Physikalische Einheit des Ist- und Sollwerts
      PhysicalQuantity { ExternalWritable := 'False'; S7_SetPoint := 'True'} : Int;   // physical quantity of the process value and setpoint / Physikalische Größe des Ist- und Sollwerts
      ActivateRecoverMode { S7_SetPoint := 'True'} : Bool := true;   // FALSE - go to inactive by error, TRUE - activate error treatment / FALSE - gehe zu Inaktiv wenn Fehler, TRUE - Fehlerbehandlung wird aktiviert
   END_VAR
   VAR RETAIN
      Warning { ExternalWritable := 'False'} : DWord;   // warning message / Anzeige von Warnungen
      WarningInternal { ExternalWritable := 'False'} : DWord;   // warning message / Anzeige von Warnungen
   END_VAR
   VAR
      Progress { ExternalWritable := 'False'} : Real;   // progress of current phase in percent / Fortschritt der aktuellen Phase in Prozent
      CurrentSetpoint { ExternalWritable := 'False'} : Real;   // current active setpoint value / Momentan wirksamer Sollwert
      CancelTuningLevel { S7_SetPoint := 'True'} : Real := 10.0;   // cancel level for setpoint change during tuning / Abschaltschwelle für Sollwertänderung während der Selbsteinstellung
      SubstituteOutput { S7_SetPoint := 'True'} : Real;   // substitute output value in case of error / Fehlerersatzausgangswert
      Config { S7_SetPoint := 'True'} : PID_CompactConfig;   // configuration data set / Struktur mit Konfigurationsdaten
      CycleTime { S7_SetPoint := 'True'} : PID_CycleTime;   // data set for cycle time estimation / Struktur mit Variablen, zur Ermittlung der Abtastzeit
      CtrlParamsBackUp { S7_SetPoint := 'True'} : PID_CompactControlParams;   // saved parameter set / Gespeicherter Parametersatz
      PIDSelfTune { S7_SetPoint := 'True'} : PID_CompactSelfTune;   // data set for self tuning / Struktur mit Variablen für die Selbsteinstellung
      PIDCtrl { S7_SetPoint := 'True'} : PID_CompactControl;   // data for controling part / Struktur für Variablen des Reglerteils
   END_VAR
   VAR RETAIN
      Retain { S7_SetPoint := 'True'} : PID_CompactRetain;   // retain data / Struktur mit Retain-Daten
   END_VAR
BEGIN
END_FUNCTION_BLOCK

DATA_BLOCK "6-ALLALARM_DB"   // DB23
VERSION : 0.1
// stored: AutoNumber true, DBAccessibleFromOPCUA true, DBAccessibleFromWebserver true, InstanceOfName B1--ALARM, InstanceOfType FB
"B1--ALARM"
BEGIN
END_DATA_BLOCK

DATA_BLOCK "A1-阀带反馈_DB"   // DB1
VERSION : 0.1
// stored: AutoNumber true, DBAccessibleFromOPCUA true, DBAccessibleFromWebserver true, InstanceOfName A1-阀带反馈, InstanceOfType FB
"A1-阀带反馈"
BEGIN
END_DATA_BLOCK

DATA_BLOCK "A14-阀反馈报警_DB"   // DB36
VERSION : 0.1
// stored: AutoNumber true, DBAccessibleFromOPCUA true, DBAccessibleFromWebserver true, InstanceOfName A14-阀反馈报警, InstanceOfType FB
"A14-阀反馈报警"
BEGIN
END_DATA_BLOCK

DATA_BLOCK "A2-阀带阀导_DB"   // DB2
VERSION : 0.1
// stored: AutoNumber true, DBAccessibleFromOPCUA true, DBAccessibleFromWebserver true, InstanceOfName A2-阀带阀导, InstanceOfType FB
"A2-阀带阀导"
BEGIN
END_DATA_BLOCK

DATA_BLOCK "A3-电机控制_DB"   // DB5
VERSION : 0.1
// stored: AutoNumber true, DBAccessibleFromOPCUA true, DBAccessibleFromWebserver true, InstanceOfName A3-电机控制, InstanceOfType FB
"A3-电机控制"
   // VAR
   //    进料泵控制 { S7_SetPoint := 'True'} : "A4-蠕动泵控制";
   //    引风频率 { S7_SetPoint := 'True'} : "A4--电机控制";
   //    送风频率 { S7_SetPoint := 'True'} : "A4--电机控制";
   //    离心雾化 { S7_SetPoint := 'True'} : "A4--电机控制";
   // END_VAR
BEGIN
END_DATA_BLOCK

DATA_BLOCK "A4-脉冲控制_DB"   // DB4
VERSION : 0.1
// stored: AutoNumber true, DBAccessibleFromOPCUA true, DBAccessibleFromWebserver true, InstanceOfName A4-脉冲控制, InstanceOfType FB
"A4-脉冲控制"
BEGIN
END_DATA_BLOCK

DATA_BLOCK "A5-模拟量输出_DB"   // DB11
VERSION : 0.1
// stored: AutoNumber true, DBAccessibleFromOPCUA true, DBAccessibleFromWebserver true, InstanceOfName A5-模拟量输出, InstanceOfType FB
"A5-模拟量输出"
BEGIN
END_DATA_BLOCK

DATA_BLOCK "A6-模拟量输入_DB"   // DB8
VERSION : 0.1
// stored: AutoNumber true, DBAccessibleFromOPCUA true, DBAccessibleFromWebserver true, InstanceOfName A6-模拟量输入, InstanceOfType FB
"A6-模拟量输入"
   // VAR
   //    进风流量计1 { S7_SetPoint := 'True'} : "0-模拟量输入";
   //    进料流量1 { S7_SetPoint := 'True'} : "0-模拟量输入";
   //    进风压差变送器1 { S7_SetPoint := 'True'} : "0-模拟量输入压差";
   //    出风压差变送器1 { S7_SetPoint := 'True'} : "0-模拟量输入压差";
   //    布袋压差变送器1 { S7_SetPoint := 'True'} : "0-模拟量输入压差";
   //    输送高效压差变送器1 { S7_SetPoint := 'True'} : "0-模拟量输入压差";
   //    进料压力1 { S7_SetPoint := 'True'} : "0-模拟量输入";
   //    塔内压力1 { S7_SetPoint := 'True'} : "0-模拟量输入";
   //    管道压力变送器1 { S7_SetPoint := 'True'} : "0-模拟量输入";
   //    进氮压力1 { S7_SetPoint := 'True'} : "0-模拟量输入";
   //    放空比例反馈1 { S7_SetPoint := 'True'} : "0-模拟量输入";
   //    进风加热比例反馈1 { S7_SetPoint := 'True'} : "0-模拟量输入";
   //    回风加热比例反馈1 { S7_SetPoint := 'True'} : "0-模拟量输入";
   //    雾化油压1 { S7_SetPoint := 'True'} : "0-模拟量输入";
   //    氧含仪11 { S7_SetPoint := 'True'} : "0-模拟量输入";
   //    氧含仪12 { S7_SetPoint := 'True'} : "0-模拟量输入";
   //    一级溶剂液位计1 { S7_SetPoint := 'True'} : "0-模拟量输入";
   //    二级溶剂液位计1 { S7_SetPoint := 'True'} : "0-模拟量输入";
   //    除雾溶剂液位计1 { S7_SetPoint := 'True'} : "0-模拟量输入";
   //    前置水罐液位1 { S7_SetPoint := 'True'} : "0-模拟量输入";
   //    阀岛气压1 { S7_SetPoint := 'True'} : "0-模拟量输入";
   //    T1S : TON_TIME;
   //    YC1 { S7_SetPoint := 'True'} : Real;
   //    延迟1 { S7_SetPoint := 'True'} : "步段延迟";
   //    延迟2 { S7_SetPoint := 'True'} : "步段延迟";
   // END_VAR
BEGIN
END_DATA_BLOCK

DATA_BLOCK "A7-温度控制_DB"   // DB13
VERSION : 0.1
// stored: AutoNumber true, DBAccessibleFromOPCUA true, DBAccessibleFromWebserver true, InstanceOfName A7-温度控制, InstanceOfType FB
"A7-温度控制"
   // VAR
   //    Modbus_Comm_Load { S7_SetPoint := 'True'} : Modbus_Comm_Load;
   //    MB_MASTER { S7_SetPoint := 'True'} : Modbus_Master;
   //    FB_DTC1 { S7_SetPoint := 'True'} : "A1-台达DTC";
   //    FB_DTC2 { S7_SetPoint := 'True'} : "A1-台达DTC";
   //    FB_DTC3 { S7_SetPoint := 'True'} : "A1-台达DTC";
   //    FB_DTC4 { S7_SetPoint := 'True'} : "A1-台达DTC";
   //    FB_DTC5 { S7_SetPoint := 'True'} : "A1-台达DTC";
   //    P { S7_SetPoint := 'True'} : Array[1..16] of Bool;
   //    R_TRIG1 : R_TRIG;
   //    FB_DTC_Instance { S7_SetPoint := 'True'} : "A1-台达DTC";
   //    FB_DTC_Instance_1 { S7_SetPoint := 'True'} : "A1-台达DTC";
   //    通信异常计数 : Array[0..16] of Int;
   //    通信故障 : Array[0..16] of Bool;
   //    总通信故障 : Bool;
   //    i : UDInt;
   // END_VAR
BEGIN
END_DATA_BLOCK

DATA_BLOCK "B2--局部连锁_DB"   // DB17
VERSION : 0.1
// stored: AutoNumber true, DBAccessibleFromOPCUA true, DBAccessibleFromWebserver true, InstanceOfName B2--局部连锁, InstanceOfType FB
"B2--局部连锁"
BEGIN
END_DATA_BLOCK

DATA_BLOCK "B3-全局连锁_DB"   // DB25
VERSION : 0.1
// stored: AutoNumber true, DBAccessibleFromOPCUA true, DBAccessibleFromWebserver true, InstanceOfName B3-全局连锁, InstanceOfType FB
"B3-全局连锁"
   // VAR
   //    T1S : TON_TIME;
   //    YC1 { S7_SetPoint := 'True'} : DInt;
   //    BJ报警上升辅助 : Bool;
   //    BJ报警下降辅助 : Bool;
   //    BJ报警上升沿 { S7_SetPoint := 'True'} : R_TRIG;
   //    BJ报警下降沿 { S7_SetPoint := 'True'} : F_TRIG;
   //    DH : Int;
   //    XT心跳上升沿延迟 : TON_TIME;
   //    XT心跳下降沿延迟 { S7_SetPoint := 'True'} : TON_TIME;
   // END_VAR
BEGIN
END_DATA_BLOCK

DATA_BLOCK "B4-清洗连锁_DB"   // DB33
VERSION : 0.1
// stored: AutoNumber true, DBAccessibleFromOPCUA true, DBAccessibleFromWebserver true, InstanceOfName B4-清洗连锁, InstanceOfType FB
"B4-清洗连锁"
BEGIN
END_DATA_BLOCK

DATA_BLOCK "C1-开式自动_DB"   // DB34
VERSION : 0.1
// stored: AutoNumber true, DBAccessibleFromOPCUA true, DBAccessibleFromWebserver true, InstanceOfName C1-开式自动, InstanceOfType FB
"C1-开式自动"
   // VAR
   //    开式自动喷雾 { S7_SetPoint := 'True'} : "开式自动喷雾块";
   //    KS开式自动自检 { S7_SetPoint := 'True'} : Bool;
   //    四参数辅助 { S7_SetPoint := 'True'} : "四参数辅助";
   //    TON1 { S7_SetPoint := 'True'} : TON_TIME;
   //    TON2 { S7_SetPoint := 'True'} : TON_TIME;
   //    TON3 { S7_SetPoint := 'True'} : TON_TIME;
   //    BD布袋反吹记录 { S7_SetPoint := 'True'} : "D3-布袋记录";
   // END_VAR
BEGIN
END_DATA_BLOCK

DATA_BLOCK "C2-闭式自动_DB"   // DB20
VERSION : 0.1
// stored: AutoNumber true, DBAccessibleFromOPCUA true, DBAccessibleFromWebserver true, InstanceOfName C2-闭式自动, InstanceOfType FB
"C2-闭式自动"
   // VAR
   //    闭式自动喷雾 { S7_SetPoint := 'True'} : "闭式自动喷雾块";
   //    雾化塔保压 { S7_SetPoint := 'True'} : "闭式保压块";
   //    TON1 { S7_SetPoint := 'True'} : TON_TIME;
   //    TON2 { S7_SetPoint := 'True'} : TON_TIME;
   //    TON3 { S7_SetPoint := 'True'} : TON_TIME;
   //    BD布袋反吹记录 { S7_SetPoint := 'True'} : "D3-布袋记录";
   //    FT1 { S7_SetPoint := 'True'} : F_TRIG;
   //    RT1 { S7_SetPoint := 'True'} : R_TRIG;
   //    RT2 { S7_SetPoint := 'True'} : R_TRIG;
   //    TP1 { S7_SetPoint := 'True'} : TP_TIME;
   // END_VAR
BEGIN
END_DATA_BLOCK

DATA_BLOCK "C3-室内CIP清洗_DB"   // DB30
VERSION : 0.1
// stored: AutoNumber true, DBAccessibleFromOPCUA true, DBAccessibleFromWebserver true, InstanceOfName C3-室内CIP清洗, InstanceOfType FB
"C3-室内CIP清洗"
   // VAR
   //    室内CIP清洗 { S7_SetPoint := 'True'} : "INCIP清洗";
   //    FT1 { S7_SetPoint := 'True'} : F_TRIG;
   //    FT2 { S7_SetPoint := 'True'} : F_TRIG;
   //    FT3 { S7_SetPoint := 'True'} : F_TRIG;
   //    TON1 { S7_SetPoint := 'True'} : TON_TIME;
   //    PT1 { S7_SetPoint := 'True'} : Time;
   //    T1S : TON_TIME;
   //    YC1 { S7_SetPoint := 'True'} : DInt;
   //    YC2 : DInt;
   //    YC3 : DInt;
   //    TP1 : Bool;
   //    TP2 : Bool;
   //    TP3 : Bool;
   //    T_10HZ : TON_TIME;
   //    GET_Instance { S7_SetPoint := 'True'} : GET;
   //    PUT_Instance { S7_SetPoint := 'True'} : PUT;
   // END_VAR
BEGIN
END_DATA_BLOCK

DATA_BLOCK "C4-室外CIP清洗_DB"   // DB31
VERSION : 0.1
// stored: AutoNumber true, DBAccessibleFromOPCUA true, DBAccessibleFromWebserver true, InstanceOfName C4-室外CIP清洗, InstanceOfType FB
"C4-室外CIP清洗"
   // VAR
   //    室外CIP清洗 { S7_SetPoint := 'True'} : "OUTCIP清洗";
   //    FT1 { S7_SetPoint := 'True'} : F_TRIG;
   //    FT2 { S7_SetPoint := 'True'} : F_TRIG;
   //    FT3 { S7_SetPoint := 'True'} : F_TRIG;
   //    TON1 { S7_SetPoint := 'True'} : TON_TIME;
   //    PT1 { S7_SetPoint := 'True'} : Time;
   //    T1S : TON_TIME;
   //    YC1 { S7_SetPoint := 'True'} : DInt;
   //    YC2 : DInt;
   //    YC3 : DInt;
   //    TP1 : Bool;
   //    TP2 : Bool;
   //    TP3 : Bool;
   //    T_10HZ : TON_TIME;
   //    GET_Instance { S7_SetPoint := 'True'} : GET;
   //    PUT_Instance { S7_SetPoint := 'True'} : PUT;
   // END_VAR
BEGIN
END_DATA_BLOCK

DATA_BLOCK "D1-室内CIP通讯_DB"   // DB32
VERSION : 0.1
// stored: AutoNumber true, DBAccessibleFromOPCUA true, DBAccessibleFromWebserver true, InstanceOfName D1-室内CIP通讯, InstanceOfType FB
"D1-室内CIP通讯"
   // VAR
   //    T_10HZ { S7_SetPoint := 'True'} : TON_TIME;
   //    FT1 { S7_SetPoint := 'True'} : F_TRIG;
   //    RT00 { S7_SetPoint := 'True'} : R_TRIG;
   //    RT10 { S7_SetPoint := 'True'} : R_TRIG;
   //    RT11 { S7_SetPoint := 'True'} : R_TRIG;
   //    RT12 { S7_SetPoint := 'True'} : R_TRIG;
   //    RT20 { S7_SetPoint := 'True'} : R_TRIG;
   //    RT21 { S7_SetPoint := 'True'} : R_TRIG;
   //    RT22 { S7_SetPoint := 'True'} : R_TRIG;
   //    RT30 { S7_SetPoint := 'True'} : R_TRIG;
   //    RT31 { S7_SetPoint := 'True'} : R_TRIG;
   //    RT32 { S7_SetPoint := 'True'} : R_TRIG;
   //    RT40 { S7_SetPoint := 'True'} : R_TRIG;
   //    RT41 { S7_SetPoint := 'True'} : R_TRIG;
   //    RT42 { S7_SetPoint := 'True'} : R_TRIG;
   //    RT50 { S7_SetPoint := 'True'} : R_TRIG;
   //    RT51 { S7_SetPoint := 'True'} : R_TRIG;
   //    RT52 { S7_SetPoint := 'True'} : R_TRIG;
   //    RT60 { S7_SetPoint := 'True'} : R_TRIG;
   //    RT61 { S7_SetPoint := 'True'} : R_TRIG;
   //    RT62 { S7_SetPoint := 'True'} : R_TRIG;
   //    RT3 { S7_SetPoint := 'True'} : R_TRIG;
   //    RS热水洗辅助 { S7_SetPoint := 'True'} : Bool;
   //    JS碱水洗辅助 : Bool;
   //    CS纯水洗辅助 : Bool;
   //    EC二纯水洗辅助 : Bool;
   //    RJ溶剂洗辅助 : Bool;
   //    PUT_Instance { S7_SetPoint := 'True'} : PUT;
   //    GET_Instance { S7_SetPoint := 'True'} : GET;
   // END_VAR
BEGIN
END_DATA_BLOCK

DATA_BLOCK "D2-室外CIP通讯_DB"   // DB35
VERSION : 0.1
// stored: AutoNumber true, DBAccessibleFromOPCUA true, DBAccessibleFromWebserver true, InstanceOfName D2-室外CIP通讯, InstanceOfType FB
"D2-室外CIP通讯"
   // VAR
   //    T_10HZ { S7_SetPoint := 'True'} : TON_TIME;
   //    FT1 { S7_SetPoint := 'True'} : F_TRIG;
   //    RT00 { S7_SetPoint := 'True'} : R_TRIG;
   //    RT10 { S7_SetPoint := 'True'} : R_TRIG;
   //    RT11 { S7_SetPoint := 'True'} : R_TRIG;
   //    RT12 { S7_SetPoint := 'True'} : R_TRIG;
   //    RT20 { S7_SetPoint := 'True'} : R_TRIG;
   //    RT21 { S7_SetPoint := 'True'} : R_TRIG;
   //    RT22 { S7_SetPoint := 'True'} : R_TRIG;
   //    RT30 { S7_SetPoint := 'True'} : R_TRIG;
   //    RT31 { S7_SetPoint := 'True'} : R_TRIG;
   //    RT32 { S7_SetPoint := 'True'} : R_TRIG;
   //    RT40 { S7_SetPoint := 'True'} : R_TRIG;
   //    RT41 { S7_SetPoint := 'True'} : R_TRIG;
   //    RT42 { S7_SetPoint := 'True'} : R_TRIG;
   //    RT50 { S7_SetPoint := 'True'} : R_TRIG;
   //    RT51 { S7_SetPoint := 'True'} : R_TRIG;
   //    RT60 { S7_SetPoint := 'True'} : R_TRIG;
   //    RT61 { S7_SetPoint := 'True'} : R_TRIG;
   //    RT62 { S7_SetPoint := 'True'} : R_TRIG;
   //    RT3 { S7_SetPoint := 'True'} : R_TRIG;
   //    RS热水洗辅助 { S7_SetPoint := 'True'} : Bool;
   //    JS碱水洗辅助 : Bool;
   //    CS纯水洗辅助 : Bool;
   //    EC二纯水洗辅助 : Bool;
   //    RJ溶剂洗辅助 : Bool;
   //    PUT_Instance { S7_SetPoint := 'True'} : PUT;
   //    GET_Instance { S7_SetPoint := 'True'} : GET;
   // END_VAR
BEGIN
END_DATA_BLOCK
